// TwinCAT 3 PLC project mobject_json
// Title: mobject-json
// Company: mobject.io
// Author: mobject dev team
// ProjectVersion: 0.5.0
// ProgramVersion: 3.1.4023.0
// libraries:
//   mobject-core, * (mobject.io)
//   Tc2_System, * (Beckhoff Automation GmbH)
//   Tc3_IotBase, * (Beckhoff Automation GmbH)
//   Tc3_JsonXml, * (Beckhoff Automation GmbH)
//   Tc3_Module, * (Beckhoff Automation GmbH)
// project tree:
//   Json Path/ I_JsonPath.TcIO, JsonPath.TcPOU
//   _Internal/JsonPath/ I_JsonPathElement.TcIO, JsonPathElement.TcPOU, JsonPathElement_ArraySingleSelector.TcPOU, JsonPathElement_Property.TcPOU, JsonPathElement_Root.TcPOU, ParseJsonPath.TcPOU

// ---- Json Path/I_JsonPath.TcIO
INTERFACE I_JsonPath

METHOD PUBLIC TryRead : HRESULT
VAR_INPUT
	Path : T_MaxString;
	Destination : ANY;
END_VAR
END_METHOD

END_INTERFACE

// ---- _Internal/JsonPath/I_JsonPathElement.TcIO
INTERFACE I_JsonPathElement EXTENDS I_Disposable

PROPERTY PUBLIC NextElement : I_JsonPathElement
GET
END_GET
SET
END_SET
END_PROPERTY

PROPERTY PUBLIC PreviousElement : I_JsonPathElement
GET
END_GET
SET
END_SET
END_PROPERTY

PROPERTY PUBLIC PropertyName : T_MAXSTRING
GET
END_GET
END_PROPERTY

METHOD PUBLIC ABSTRACT ResolveToSJsonValue : SJsonValue
VAR_INPUT
	jsonParser : REFERENCE TO FB_JsonDomParser;
	jsonDocument : SJsonValue;
END_VAR
END_METHOD

END_INTERFACE

// ---- Json Path/JsonPath.TcPOU
{attribute 'linkalways'} 
{attribute 'no_explicit_call' := 'This FB is a CLASS and must be accessed using methods or properties'}
{attribute 'enable_dynamic_creation'}
FUNCTION_BLOCK JsonPath IMPLEMENTS I_JsonPath
VAR
	jsonParser : FB_JsonDomParser;
	jsonDocument : SJsonValue;
END_VAR

METHOD PUBLIC Parse : I_JsonPath
VAR_INPUT
	JsonString : REFERENCE TO STRING;
END_VAR
jsonDocument := jsonParser.ParseDocument(JsonString);
Parse := this^;
END_METHOD

METHOD PUBLIC ParseFromHttpRequest : I_JsonPath
VAR_INPUT
	HttpRequest : REFERENCE TO FB_IotHttpRequest;
END_VAR
jsonDocument := HttpRequest.GetJsonDomContent(jsonParser);
ParseFromHttpRequest := this^;
END_METHOD

METHOD PUBLIC TryRead : HRESULT
VAR_INPUT
	Path : T_MaxString;
	Destination : ANY;
END_VAR
VAR
	result : HRESULT;
	jsonElement : I_JsonPathElement;
	jsonValue : SJsonValue;
	_BOOL : BOOL;
	_DINT : DINT;
	_LINT : LINT;
	_UDINT : UDINT;
	_ULINT : ULINT;
	_LREAL : LREAL;
	_STRING : POINTER TO STRING(1);
END_VAR
ParseJsonPath(Path,jsonElement);

IF FAILED(result) THEN
	TryRead := result;
	RETURN;
END_IF

jsonValue := jsonElement.ResolveToSJsonValue(jsonParser,jsonDocument);
jsonElement.Release();

IF jsonValue = 0 THEN
	TryRead := NOT_FOUND;
	RETURN;
END_IF

IF jsonParser.IsBool(jsonValue) THEN
	_BOOL := jsonParser.GetBool(jsonValue);
	TryRead := Convert_BOOL_TO_(_BOOL,Destination);
	RETURN;
END_IF

IF jsonParser.IsInt(jsonValue) THEN
	_DINT := jsonParser.GetInt(jsonValue);
	TryRead := Convert_DINT_TO_(_DINT,Destination);
	RETURN;
END_IF

IF jsonParser.IsInt64(jsonValue) THEN
	_LINT := jsonParser.GetInt64(jsonValue);
	TryRead := Convert_LINT_TO_(_LINT,Destination);
	RETURN;
END_IF

IF jsonParser.IsUInt(jsonValue) THEN
	_UDINT := jsonParser.GetUInt(jsonValue);
	TryRead := Convert_UDINT_TO_(_UDINT,Destination);
	RETURN;
END_IF

IF jsonParser.IsUInt64(jsonValue) THEN
	_ULINT := jsonParser.GetUInt64(jsonValue);
	TryRead := Convert_ULINT_TO_(_ULINT,Destination);
	RETURN;
END_IF

IF jsonParser.IsDouble(jsonValue) THEN
	_LREAL := jsonParser.GetDouble(jsonValue);
	TryRead := Convert_LREAL_TO_(_LREAL,Destination);
	RETURN;
END_IF

IF jsonParser.IsString(jsonValue) AND Destination.TypeClass = __SYSTEM.TYPE_CLASS.TYPE_STRING THEN
	_STRING := Destination.pValue;
	IF (jsonParser.CopyString(jsonValue,_STRING^,Destination.diSize) > 0) THEN;
		TryRead := S_OK;
		RETURN;
	END_IF
END_IF
END_METHOD

END_FUNCTION_BLOCK

// ---- _Internal/JsonPath/ParseJsonPath.TcPOU
FUNCTION ParseJsonPath : I_JsonPathElement
VAR_INPUT
	Path : REFERENCE TO STRING;
	JsonPathElement : REFERENCE TO I_JsonPathElement;
END_VAR
VAR
	pRootElement : POINTER TO JsonPathElement_Root;
	pPropertyElement : POINTER TO JsonPathElement_Property; 
	pArrayElement : POINTER TO JsonPathElement_ArraySingleSelector; 
	
	lastElement : I_JsonPathElement;
	parsePosition : UDINT;
	
	currentlyParsing : (NOTHING, DOT_NOTATION_PROPERTY, BRACKET_NOTATION_PROPERTY_OR_ARRAY, BRACKET_NOTATION_PROPERTY_ELEMENT, BRACKET_NOTATION_ARRAY_ELEMENT);
	
	currentElementStart : UDINT;
	currentElementEnd : UDINT;
	currentElementLength : UDINT;
	elementText : T_MAXSTRING;
	endOfRepeat : BOOL;
END_VAR
VAR CONSTANT
	PERIOD : BYTE := 16#2E; // .
	DOLLAR_SIGN : BYTE := 16#24; // $
	SINGLE_QUOTE : BYTE := 16#27; // '
	LEFT_SQUARE_BRACKET : BYTE := 16#5B; // [
	RIGHT_SQUARE_BRACKET : BYTE := 16#5D; // ]
	NULL : BYTE := 0; // null
END_VAR

IF JsonPathElement <> 0 THEN
	JsonPathElement.Release();
END_IF

pRootElement := __NEW(JsonPathElement_Root(PreviousElement := 0,NextElement := 0));
lastElement := pRootElement^;

IF Path[0] = NULL THEN
	JsonPathElement := lastElement;
	RETURN;
END_IF

parsePosition := 0;
currentlyParsing := NOTHING;

REPEAT 
	
	IF Path[parsePosition] = NULL THEN
		 endOfRepeat := TRUE;
	END_IF
		
	CASE currentlyParsing OF
		
		NOTHING: 
		
			IF Path[parsePosition] = DOLLAR_SIGN THEN
				// No action
				
			ELSIF Path[parsePosition] = PERIOD THEN
				// No action
				
			ELSIF Path[parsePosition] = LEFT_SQUARE_BRACKET THEN
				currentlyParsing := BRACKET_NOTATION_PROPERTY_OR_ARRAY;				
				
			ELSIF Path[parsePosition] = RIGHT_SQUARE_BRACKET THEN
				// No action
				
			ELSIF Path[parsePosition] = SINGLE_QUOTE THEN
				// No action
				
			ELSE
				currentlyParsing := DOT_NOTATION_PROPERTY;
				currentElementStart := parsePosition;			
			END_IF
			
		DOT_NOTATION_PROPERTY:
		
			IF Path[parsePosition] = PERIOD  OR Path[parsePosition] = LEFT_SQUARE_BRACKET OR Path[parsePosition] = NULL THEN
				
				currentElementEnd := parsePosition - 1;
				
				currentElementLength := 1 + currentElementEnd - currentElementStart;
				memset(ADR(elementText),0,SIZEOF(elementText));
				memcpy(ADR(elementText),ADR(Path[currentElementStart]),currentElementLength);
				
				pPropertyElement := __NEW(JsonPathElement_Property(PreviousElement := 0,NextElement := 0, Name := elementText));
				lastElement.NextElement := pPropertyElement^;
				lastElement	:= pPropertyElement^;
						
				currentlyParsing := NOTHING;
				CONTINUE;
				
			END_IF
			
		BRACKET_NOTATION_PROPERTY_OR_ARRAY:
		
			IF Path[parsePosition] = SINGLE_QUOTE THEN
				currentlyParsing := BRACKET_NOTATION_PROPERTY_ELEMENT;
				currentElementStart := parsePosition + 1;			
			ELSE
				currentlyParsing := BRACKET_NOTATION_ARRAY_ELEMENT;
				currentElementStart := parsePosition;			
			END_IF
			
		BRACKET_NOTATION_PROPERTY_ELEMENT:
		
			IF Path[parsePosition] = SINGLE_QUOTE THEN
				
				currentElementEnd := parsePosition - 1;

				currentElementLength := 1 + currentElementEnd - currentElementStart;
				memset(ADR(elementText),0,SIZEOF(elementText));
				memcpy(ADR(elementText),ADR(Path[currentElementStart]),currentElementLength);
				
				pPropertyElement := __NEW(JsonPathElement_Property(PreviousElement := 0,NextElement := 0, Name := elementText));
				lastElement.NextElement := pPropertyElement^;
				lastElement	:= pPropertyElement^;
				
				currentlyParsing := NOTHING;
						
			END_IF
			
		BRACKET_NOTATION_ARRAY_ELEMENT:
		
			IF Path[parsePosition] = RIGHT_SQUARE_BRACKET THEN
				
				currentElementEnd := parsePosition - 1;
				
				currentElementLength := 1 + currentElementEnd - currentElementStart;
				memset(ADR(elementText),0,SIZEOF(elementText));
				memcpy(ADR(elementText),ADR(Path[currentElementStart]),currentElementLength);
				
				pArrayElement := __NEW(JsonPathElement_ArraySingleSelector(PreviousElement := 0,NextElement := 0, IndexString := elementText));
				lastElement.NextElement := pArrayElement^;
				lastElement	:= pArrayElement^;
				
				currentlyParsing := NOTHING;
						
			END_IF
			

	END_CASE
	
	parsePosition := parsePosition + 1;
	
UNTIL endOfRepeat 
END_REPEAT
	
JsonPathElement := lastElement;

END_FUNCTION

// ---- _Internal/JsonPath/JsonPathElement.TcPOU
{attribute 'linkalways'} 
{attribute 'no_explicit_call' := 'This FB is a CLASS and must be accessed using methods or properties'}
{attribute 'enable_dynamic_creation'}
FUNCTION_BLOCK ABSTRACT JsonPathElement EXTENDS Disposable IMPLEMENTS I_JsonPathElement
VAR
	_previousElement, _nextElement : I_JsonPathElement;
END_VAR

METHOD AddReference
VAR_INPUT
END_VAR
IF NextElement <> 0 THEN
	NextElement.AddReference();
END_IF

SUPER^.AddReference();
END_METHOD

METHOD FB_init : BOOL
VAR_INPUT
	bInitRetains : BOOL; // if TRUE, the retain variables are initialized (warm start / cold start)
	bInCopyCode : BOOL;  // if TRUE, the instance afterwards gets moved into the copy code (online change)
	PreviousElement : I_JsonPathElement;
	NextElement : I_JsonPathElement; 
END_VAR
THIS^._previousElement := PreviousElement;
THIS^._nextElement := NextElement;
END_METHOD

PROPERTY PUBLIC NextElement : I_JsonPathElement
GET
NextElement := _nextElement;
END_GET
SET
VAR
	self : I_JsonPathElement;
END_VAR
_nextElement := NextElement;

IF NextElement = 0 THEN
	RETURN;
END_IF

self := THIS^;

IF NextElement.PreviousElement <> self THEN
	NextElement.PreviousElement := self;
END_IF;
END_SET
END_PROPERTY

PROPERTY PUBLIC PreviousElement : I_JsonPathElement
GET
PreviousElement := _previousElement;
END_GET
SET
VAR
	self : I_JsonPathElement;
END_VAR
_previousElement := PreviousElement;

IF PreviousElement = 0 THEN
	RETURN;
END_IF

self := THIS^;

IF PreviousElement.NextElement <> self THEN
	PreviousElement.NextElement := self;
END_IF;
END_SET
END_PROPERTY

PROPERTY PUBLIC ABSTRACT PropertyName : T_MAXSTRING
GET
END_GET
END_PROPERTY

METHOD Release
VAR_INPUT
END_VAR
IF PreviousElement <> 0 THEN
	PreviousElement.NextElement := 0;
	PreviousElement.Release();
END_IF

IF NextElement <> 0 THEN
	NextElement.PreviousElement := 0;
	NextElement.Release();
END_IF

SUPER^.Release();
END_METHOD

METHOD PUBLIC ABSTRACT ResolveToSJsonValue : SJsonValue
VAR_INPUT
	jsonParser : REFERENCE TO FB_JsonDomParser;
	jsonDocument : SJsonValue;
END_VAR
END_METHOD

END_FUNCTION_BLOCK

// ---- _Internal/JsonPath/JsonPathElement_Root.TcPOU
{attribute 'linkalways'} 
{attribute 'no_explicit_call' := 'This FB is a CLASS and must be accessed using methods or properties'}
{attribute 'enable_dynamic_creation'}
FUNCTION_BLOCK JsonPathElement_Root EXTENDS JsonPathElement 
VAR
END_VAR

PROPERTY PUBLIC PropertyName : T_MAXSTRING
GET
PropertyName := 'root';
END_GET
END_PROPERTY

METHOD PUBLIC ResolveToSJsonValue : SJsonValue
VAR_INPUT
	jsonParser : REFERENCE TO FB_JsonDomParser;
	jsonDocument : SJsonValue;
END_VAR
ResolveToSJsonValue := jsonDocument;
END_METHOD

END_FUNCTION_BLOCK

// ---- _Internal/JsonPath/JsonPathElement_Property.TcPOU
{attribute 'linkalways'} 
{attribute 'no_explicit_call' := 'This FB is a CLASS and must be accessed using methods or properties'}
{attribute 'enable_dynamic_creation'}
FUNCTION_BLOCK JsonPathElement_Property EXTENDS JsonPathElement 
VAR
	name : T_MAXSTRING;
END_VAR

METHOD FB_init : BOOL
VAR_INPUT
	bInitRetains : BOOL; // if TRUE, the retain variables are initialized (warm start / cold start)
	bInCopyCode : BOOL;  // if TRUE, the instance afterwards gets moved into the copy code (online change)
	PreviousElement : I_JsonPathElement;
	NextElement : I_JsonPathElement; 
	Name : T_MAXSTRING;
END_VAR
This^.name := Name;
END_METHOD

PROPERTY PUBLIC PropertyName : T_MAXSTRING
GET
PropertyName := name;
END_GET
END_PROPERTY

METHOD PUBLIC ResolveToSJsonValue : SJsonValue
VAR_INPUT
	jsonParser : REFERENCE TO FB_JsonDomParser;
	jsonDocument : SJsonValue;
END_VAR
VAR
	currentPosition : SJsonValue;
	memberPath : SJsonValue;
END_VAR
IF PreviousElement <> 0 THEN
	currentPosition := PreviousElement.ResolveToSJsonValue(jsonParser,jsonDocument);
ELSE
	currentPosition := jsonDocument;
END_IF

IF currentPosition = 0 THEN
	RETURN;
END_IF

ResolveToSJsonValue := jsonParser.FindMember(currentPosition,name);
END_METHOD

END_FUNCTION_BLOCK

// ---- _Internal/JsonPath/JsonPathElement_ArraySingleSelector.TcPOU
{attribute 'linkalways'} 
{attribute 'no_explicit_call' := 'This FB is a CLASS and must be accessed using methods or properties'}
{attribute 'enable_dynamic_creation'}
FUNCTION_BLOCK JsonPathElement_ArraySingleSelector EXTENDS JsonPathElement 
VAR
	_index : UDINT;
END_VAR

METHOD FB_init : BOOL
VAR_INPUT
	bInitRetains : BOOL; // if TRUE, the retain variables are initialized (warm start / cold start)
	bInCopyCode : BOOL;  // if TRUE, the instance afterwards gets moved into the copy code (online change)
	PreviousElement : I_JsonPathElement;
	NextElement : I_JsonPathElement; 
	IndexString : String;
END_VAR
This^._index := STRING_TO_UDINT(IndexString);
END_METHOD

PROPERTY PUBLIC Index : UDINT
GET
Index := _index;
END_GET
END_PROPERTY

PROPERTY PUBLIC PropertyName : T_MAXSTRING
GET
IF PreviousElement = 0 THEN
	RETURN;	
END_IF

PropertyName := PreviousElement.PropertyName;
END_GET
END_PROPERTY

METHOD PUBLIC ResolveToSJsonValue : SJsonValue
VAR_INPUT
	jsonParser : REFERENCE TO FB_JsonDomParser;
	jsonDocument : SJsonValue;
END_VAR
VAR
	currentPosition : SJsonValue;
END_VAR
IF PreviousElement <> 0 THEN
	currentPosition := PreviousElement.ResolveToSJsonValue(jsonParser,jsonDocument);
ELSE
	currentPosition := jsonDocument;
END_IF

IF currentPosition = 0 THEN
	RETURN;
END_IF

ResolveToSJsonValue := jsonParser.GetArrayValueByIdx(currentPosition, Index);
END_METHOD

END_FUNCTION_BLOCK
